Staubli VAL3: Axis7onPosition.pgx

public program Axis7onPosition(num x_nPos (dimensions=1), num x_nPrecent (dimensions=1), bool& x_bOK (dimensions=1))
  local num l_nNum
begin

  x_bOK=false
  call GetAxis7Pos(l_nNum,x_nPrecent)
  x_bOK=abs(l_nNum-x_nPos)<0.001

end
